FUNCTION GetLastSegmentFromNamespace : T_MAXSTRING
VAR_INPUT
	Symbol : T_MAXSTRING;
END_VAR
VAR
	splitNamespace : t_MAXSTRING;
END_VAR

FindAndSplitChar( 
	sSeparatorChar := '.',  
	pSrcString := ADR(Symbol),                                  
	pLeftString := ADR(splitNamespace),   
	nLeftSize := SIZEOF(splitNamespace),                                  
	pRightString := ADR(GetLastSegmentFromNamespace), 
	nRightSize := SIZEOF(GetLastSegmentFromNamespace),                                
	bSearchFromRight := TRUE 
);

END_FUNCTION

(* stored: Version 1.1.0.1, ProductVersion 3.1.4024.12
   POU GetLastSegmentFromNamespace: Id {d6d8744b-93cf-0c85-19a8-46b457979426}, SpecialFunc None *)
